PROGRAM PRG_2_PMPS
VAR
    fbArbiterIO: FB_SubSysToArbiter_IO;
END_VAR

GVL_PMPS.fbFastFaultOutput1.Execute(i_xVeto := (PMPS_GVL.stCurrentBeamParameters.aVetoDevices[PMPS.K_Stopper.MR1K1_OUT]
                                      AND NOT PMPS_GVL.stCurrentBeamParameters.aVetoDevices[PMPS.K_Stopper.MR1K1_IN])
                                       OR PMPS_GVL.stCurrentBeamParameters.aVetoDevices[PMPS.K_Stopper.ST1K2]);
GVL_PMPS.fbFastFaultOutput2.Execute();

//Code for Requesting full beam arbitration
fbArbiter.AddRequest(nReqID := 16#FAFA, stReqBp := PMPS_GVL.cstFullBeam, sDevName := 'plc-qrix-vac');
fbArbiterIO(
	i_bVeto := (PMPS_GVL.stCurrentBeamParameters.aVetoDevices[PMPS.K_Stopper.MR1K1_OUT]
                                      AND NOT PMPS_GVL.stCurrentBeamParameters.aVetoDevices[PMPS.K_Stopper.MR1K1_IN])
                                       OR PMPS_GVL.stCurrentBeamParameters.aVetoDevices[PMPS.K_Stopper.ST1K2],
    Arbiter:=GVL_PMPS.fbArbiter,
    fbFFHWO:=GVL_PMPS.fbFastFaultOutput1);

END_PROGRAM

(* stored: Version 1.1.0.1, ProductVersion 3.1.4022.18
   POU PRG_2_PMPS: Id {b84dea55-5b52-40eb-8f1a-0d90375bdbc2}, SpecialFunc None *)
